// TIA Portal V17 export
// export: Created 2022-07-20T07:02:35.7949901Z, ExportSetting WithDefaults, DisplayName Totally Integrated Automation Portal, DisplayVersion V17, DisplayName TIA Portal Openness, DisplayVersion V17, DisplayName TIA Portal Version Control Interface, DisplayVersion V17, DisplayName SINAMICS Startdrive Advanced, DisplayVersion V17, DisplayName SINAMICS Startdrive G130, G150, S120, S150, SINAMICS MV, S210, DisplayVersion V17, DisplayName SINAMICS Startdrive G110M, G120, G120C, G120D, G120P, G115D, DisplayVersion V17, DisplayName STEP 7 Professional, DisplayVersion V17, DisplayName STEP 7 Safety, DisplayVersion V17, DisplayName WinCC Advanced, DisplayVersion V17
VAR_GLOBAL   // PLC tag table "UserDiag_Constants"
END_VAR
VAR_GLOBAL CONSTANT   // user constants
   USERDIAG_IOSYSTEM_1 : Int := 1;   // Index for first IO-System/DP-Mastersystem
   USERDIAG_IOSYSTEM_2 : Int := 2;   // Index for second IO-System/DP-Mastersystem
   USERDIAG_DEVICES_PER_SCREEN_UPPER_LIM : Int := 32;   // Upper limit of devices per HMI screen
   USERDIAG_SLOTS_PER_SCREEN_UPPER_LIM : Int := 31;   // Upper limit of slots per HMI screen
   USERDIAG_SLOTS_PER_DEVICE_UPPER_LIM : Int := 31;   // max number of modules per device
   USERDIAG_DEVICES_PER_IO_SYSTEM_UPPER_LIM : Int := 128;   // Upper limit of devices/slaves per IO-System/DP-Mastersystem
   USERDIAG_SLOTS_PER_PLC_UPPER_LIM : Int := 31;   // max number of local modules
   USERDIAG_IO_SYSTEMS_UPPER_LIM : Int := 2;   // Upper limit of IO-Systems/DP-Mastersystems
END_VAR
